{attribute addProperty BoxType "EL3602-0000-0016"}
{attribute addProperty Id "UnderrangeAT %I*BOOL811OverrangeAT %I*BOOL812Limit_xAT %I*ARRAY[0 ..1] OF BYTE1620ErrorAT %I*BOOL817TxPDO_StateAT %I*BOOL817TxPDO_ToggleAT %I*BOOL819ValueAT %I*DINT32417"}
{attribute addProperty CRC "3186111617"}
{attribute addProperty SizeInBites "88"}
{attribute addProperty SizeInBytes "11"}
TYPE AI_Inputs_Channel_513C0694 :
STRUCT
	{attribute addProperty Name "Underrange"}
	Underrange AT %I* : BOOL;
	{attribute addProperty Name "Overrange"}
	Overrange AT %I* : BOOL;
	{attribute addProperty Name "Limit"}
	Limit_x AT %I* : ARRAY[0 ..1] OF BYTE;
	{attribute addProperty Name "Error"}
	Error AT %I* : BOOL;
	{attribute addProperty Name "TxPDO_State"}
	TxPDO_State AT %I* : BOOL;
	{attribute addProperty Name "TxPDO_Toggle"}
	TxPDO_Toggle AT %I* : BOOL;
	{attribute addProperty Name "Value"}
	Value AT %I* : DINT;
END_STRUCT
END_TYPE

(* stored: Version 1.2.0.0, ProductVersion 3.1.4024.9
   DUT AI_Inputs_Channel_513C0694: Id {bf575770-7408-43af-9345-9227584ac4fb} *)
